PROGRAM MAIN
VAR
END_VAR

Lichtsturing();
EnOcean();
Beamercontrol();
Tcp_ip();

END_PROGRAM

(* stored: Version 1.1.0.1, ProductVersion 3.1.4022.10
   POU MAIN: Id {6a06684d-bcf5-416c-bb0a-1c04413e8cd7}, SpecialFunc None *)
